(* CODESYS project Buffer Station - Costa v5.0.project

Project tree, tasks and I/O mapping:
  Device : CODESYS Control Win V3, 3S - Smart Software Solutions GmbH, order no. 305021, version 3.5.11.30
    application Application
      libraries: Standard, * (System)
      task MainTask (cyclic, interval t#20ms, priority 1) calls PLC_PRG
      program PLC_PRG [LD]: A_Reset_Geral
      Symbols
*)

// Device/Application/PLC_PRG
PROGRAM PLC_PRG
VAR
	// Entradas
	firstScan		: BOOL := TRUE; // Ela nasce ligada
	Remover_Plastico	: BOOL := TRUE;
	Remover_Metal		: BOOL := TRUE;
	M_P0_Home: INT;
	xStart_Button: BOOL;
	M_P1_Alimentacao: INT;
	
	S_Capacitivo: BOOL;
	S_Indutivo: BOOL;
	Emitter: BOOL;
	Conveyor_Motor: INT;
	M_P2_Ident: INT;
	S_T4_Metal_Out: BOOL;
	T2_Wait_Pos: TIME;
	tonPos: TON;
	M_P3_Desvia_Plastico: INT;
	Pusher: BOOL;
	M_P4_Pusher_OFF: INT;
	xReset_Button: BOOL;
	xStop_Button: BOOL;
	S_T3_Pla_Out: BOOL;
	trigReset: R_TRIG;
	aux1: BOOL;
END_VAR
VAR // added by the converter: edge detectors and wires of the graphical bodies
    _w1, _w2, _w3, _w4, _w5, _w6, _w7 : BOOL;
    _ft1 : F_TRIG;
END_VAR

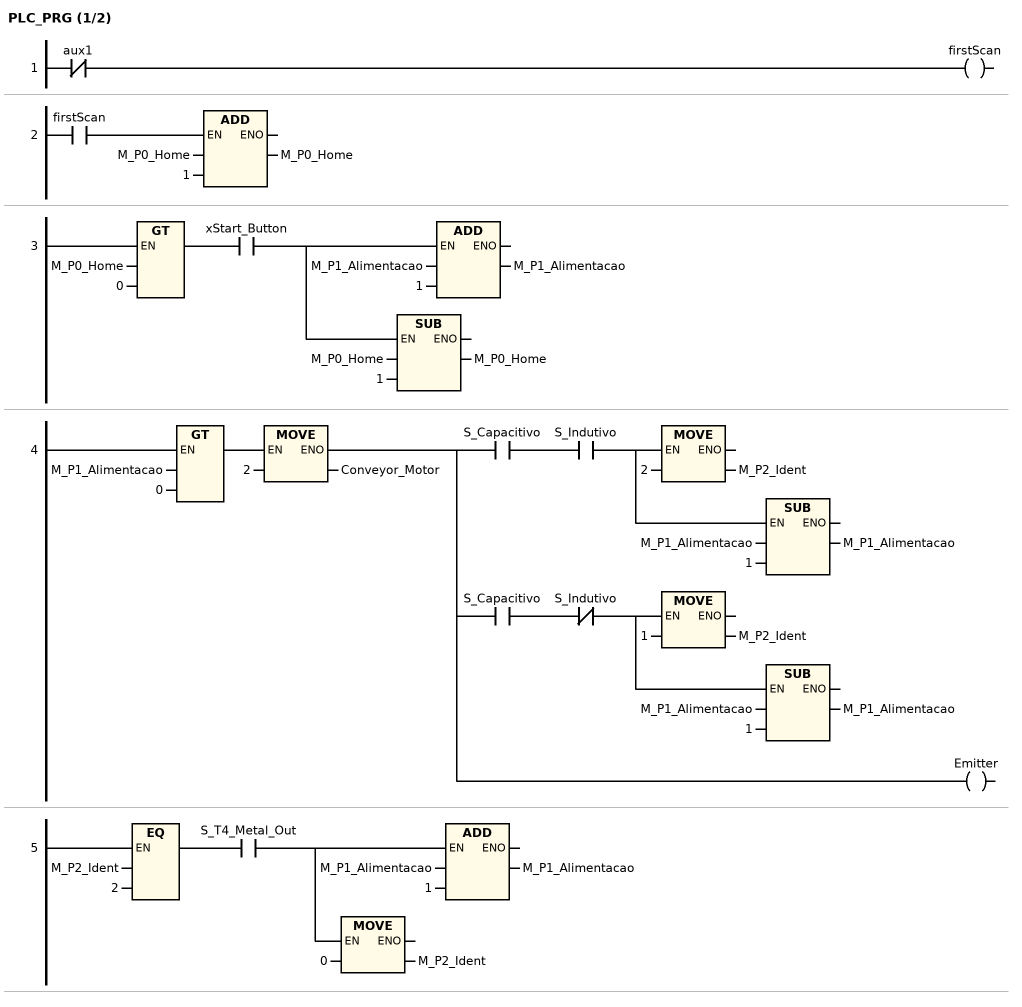
// NETWORK 1
firstScan := NOT aux1;

// NETWORK 2
IF firstScan THEN M_P0_Home := M_P0_Home + 1; END_IF

// NETWORK 3
_w1 := M_P0_Home > 0 AND xStart_Button;
IF _w1 THEN M_P1_Alimentacao := M_P1_Alimentacao + 1; END_IF
IF _w1 THEN M_P0_Home := M_P0_Home - 1; END_IF

// NETWORK 4
_w2 := M_P1_Alimentacao > 0;
IF _w2 THEN Conveyor_Motor := 2; END_IF
_w3 := _w2 AND S_Capacitivo AND S_Indutivo;
IF _w3 THEN M_P2_Ident := 2; END_IF
IF _w3 THEN M_P1_Alimentacao := M_P1_Alimentacao - 1; END_IF
_w4 := _w2 AND S_Capacitivo AND NOT S_Indutivo;
IF _w4 THEN M_P2_Ident := 1; END_IF
IF _w4 THEN M_P1_Alimentacao := M_P1_Alimentacao - 1; END_IF
Emitter := _w2;

// NETWORK 5
_w5 := M_P2_Ident = 2 AND S_T4_Metal_Out;
IF _w5 THEN M_P1_Alimentacao := M_P1_Alimentacao + 1; END_IF
IF _w5 THEN M_P2_Ident := 0; END_IF

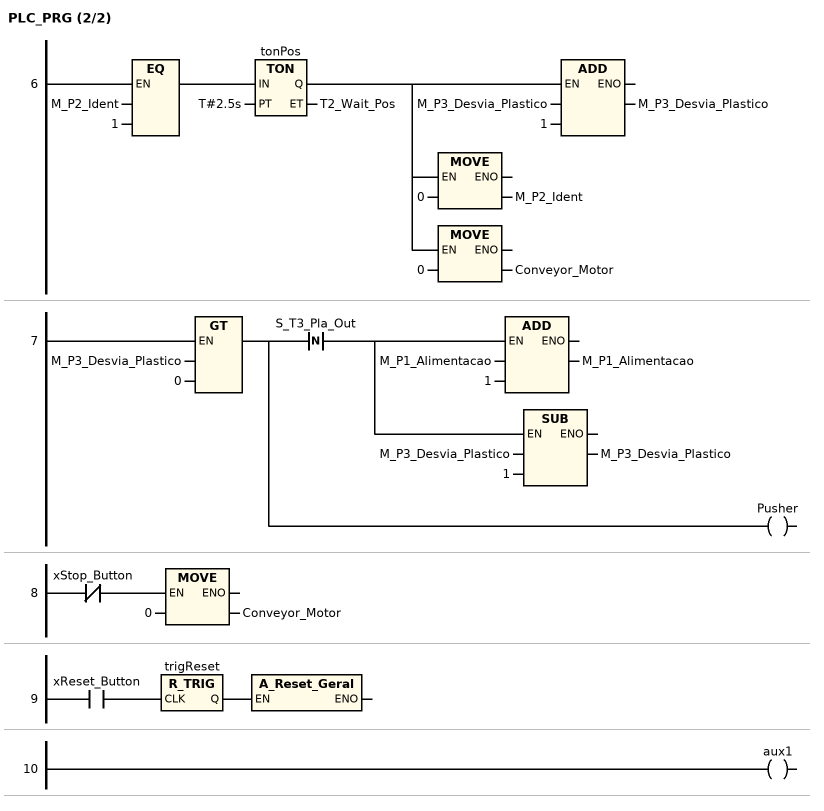
// NETWORK 6
tonPos(IN := M_P2_Ident = 1, PT := T#2.5s, ET => T2_Wait_Pos); // TON
IF tonPos.Q THEN M_P3_Desvia_Plastico := M_P3_Desvia_Plastico + 1; END_IF
IF tonPos.Q THEN M_P2_Ident := 0; END_IF
IF tonPos.Q THEN Conveyor_Motor := 0; END_IF

// NETWORK 7
_w6 := M_P3_Desvia_Plastico > 0;
_ft1(CLK := S_T3_Pla_Out);
_w7 := _w6 AND _ft1.Q;
IF _w7 THEN M_P1_Alimentacao := M_P1_Alimentacao + 1; END_IF
IF _w7 THEN M_P3_Desvia_Plastico := M_P3_Desvia_Plastico - 1; END_IF
Pusher := _w6;

// NETWORK 8
IF NOT xStop_Button THEN Conveyor_Motor := 0; END_IF

// NETWORK 9
trigReset(CLK := xReset_Button); // R_TRIG
IF trigReset.Q THEN A_Reset_Geral(); END_IF

// NETWORK 10
aux1 := TRUE;

ACTION A_Reset_Geral:
// --- ESTADO INICIAL DO SISTEMA ---
Remover_Plastico := TRUE;   //
Remover_Metal    := TRUE;   //

// --- RESET DOS LUGARES (TOKENS DA REDE DE PETRI - TIPO INT) ---
M_P0_Home            := 1;  // Marcação inicial: o token volta para o início
M_P1_Alimentacao     := 0;  //
M_P2_Ident           := 0;  //
M_P3_Desvia_Plastico := 0;  //
M_P4_Pusher_OFF      := 0;  //

// --- RESET DE BITS DE TRANSIÇÃO E LÓGICA (BOOL) ---
xStart_Button       := FALSE;    //
S_T4_Metal_Out := FALSE;    //
S_T3_Pla_Out  := FALSE;    //

// --- RESET DE SAÍDAS E ATUADORES ---
Conveyor_Motor := 0;        // Motor parado (INT)
Pusher         := FALSE;    // Pistão recolhido
Emitter        := FALSE;    // Gerador de peças desligado

// --- RESET DE TIMERS ---
tonPos(IN := FALSE);       // Garante que o cronômetro volte ao zero
END_ACTION

END_PROGRAM
